ABB RobotStudio station: step_smartcomponet_20200824-230958.rsstn

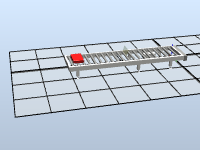
Station step_smartcomponet (saved by RobotStudio 6.8.8307.1040)
Controller IRB_120_3kg_0.58m_3
Layout (positions relative to the parent item):
  - IRB4600_60_205_C_01 [mechanism, from Robots\IRB4600_60_205_C_G_01.rslib] at (0, 0, 0) mm; joint values [0, 0, 0, 0, 0.5236, 0] (rad or m)
  - 950_4000_h2 [part, from Equipment\Conveyor 950 4000 h2.rslib]
  - CAJA [part, from Step_vacum_gripper\SOLCAJA.rslib] at (2900, 450, 412.42) mm
  - SmartComponent_1 [smart component]
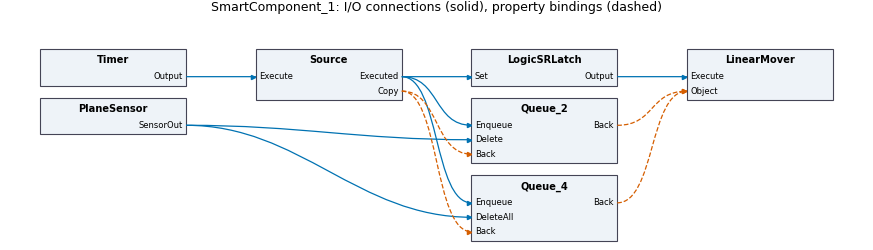
      connections:
        Timer.Output -> Source.Execute
        Source.Executed -> Queue_2.Enqueue
        LogicSRLatch.Output -> LinearMover.Execute
        PlaneSensor.SensorOut -> Queue_2.Delete
        Source.Executed -> Queue_4.Enqueue
        PlaneSensor.SensorOut -> Queue_4.DeleteAll
        Source.Executed -> LogicSRLatch.Set
        Source.Copy => Queue_2.Back
        Queue_2.Back => LinearMover.Object
        Source.Copy => Queue_4.Back
        Queue_4.Back => LinearMover.Object
    - Source [smart component, from Components\Source.rslib]
        properties: Source=CAJA; Copy=(none); Parent=(none); Position=[3.9 0.76 0.464418]; Orientation=[0 0 0]; Transient=true; PhysicsBehavior=0
    - Timer [smart component, from Components\Timer.rslib]
        properties: StartTime=0; Interval=7; Repeat=true; CurrentTime=39.312
    - LinearMover [smart component, from Components\LinearMover.rslib]
        properties: Object=(none); Direction=[-1 0 0]; Speed=0.6; Reference=Global; ReferenceObject=(none)
    - PlaneSensor [smart component, from Components\PlaneSensor.rslib]
        properties: Origin=[2 0.1 0.45]; Axis1=[0 0.2 0.3]; Axis2=[0 0.5 0]; SensedPart=(none)
      - _sensorPart_ [part]
    - LogicSRLatch [smart component, from Components\LogicSRLatch.rslib]
    - Queue_4 [smart component, from Components\Queue.rslib]
        properties: Back=(none); Front=(none); Queue=; NumberOfObjects=0
